FUNCTION_BLOCK FB_ModeVisu IMPLEMENTS I_Mode
VAR_INPUT
END_VAR
VAR_OUTPUT
END_VAR
VAR
END_VAR

METHOD Auto
VAR_INPUT
	bEnable : BOOL;
END_VAR
IF bEnable THEN 
	HMI.eMode := E_Mode.Auto;
END_IF
END_METHOD

METHOD Manual
VAR_INPUT
	bEnable: BOOL;
END_VAR
IF bEnable THEN 
	HMI.eMode := E_Mode.Manual;
END_IF
END_METHOD

METHOD OFF
VAR_INPUT
	bEnable: BOOL;
END_VAR
IF bEnable THEN 
	HMI.eMode := E_Mode.OFF;
END_IF
END_METHOD

END_FUNCTION_BLOCK

(* stored: Version 1.1.0.1, ProductVersion 3.1.4024.12
   POU FB_ModeVisu: Id {fa1ca2fb-23cc-4093-984f-ae1fb5ab29a5}, SpecialFunc None
   Method Auto: Id {09186efb-5f05-45f5-adc8-b7938cc6a484}
   Method Manual: Id {c6924fcd-4e1a-4c1d-94ef-c2847d6bb2d0}
   Method OFF: Id {31a10150-8af5-42cb-a52e-e19248c6a30f} *)
